(*
Signals are sent only once.
In order to resend the same signal, a global or a local reset is necessary.
*)
FUNCTION_BLOCK SignalHandling EXTENDS ExceptionHandling IMPLEMENTS I_SignalHandling 
VAR_OUTPUT
END_VAR

VAR_STAT
	bResetSignals : BOOL;
	aSignals : ARRAY[1..cMaxNumSignals] OF ST_Signal;
	uiSignalCounter : UINT := 0;
END_VAR

VAR CONSTANT
	cMaxNumSignals : UINT := 200;
	aEmptySignals : ARRAY[1..cMaxNumSignals] OF ST_Signal;
END_VAR

SUPER^();

METHOD BuildSignal : ST_Signal
VAR_INPUT
	eSignal	: E_Signal;
END_VAR
BuildSignal.eSignal := eSignal;
BuildSignal.eSignalOrigin := getSignalOrigin;
BuildSignal.sTimestamp := SYSTEMTIME_TO_STRING(fbTime.systemTime);
END_METHOD

METHOD GenericReceive : BOOL
VAR_INPUT
	eSignal : E_Signal;
END_VAR
VAR
	i : UINT;
END_VAR
FOR i := 1 TO uiSignalCounter
DO

	IF aSignals[i].eSignal = eSignal
	THEN
		//Reset the signal now
		GenericReceive := TRUE;
		RETURN;
	END_IF
		
END_FOR
END_METHOD

{warning 'Eigenschaftenimplementierung hinzufügen'}
PROPERTY getSignal : ST_Signal
GET
VAR CONSTANT
	stEmptySignal : ST_Signal;
END_VAR
IF SignalAvailable()
THEN
	getSignal := aSignals[uiSignalCounter];
	aSignals[uiSignalCounter] := stEmptySignal;
	uiSignalCounter := uiSignalCounter - 1;
END_IF
END_GET
END_PROPERTY

PROPERTY getSignalOrigin : E_Origin
GET
getSignalOrigin := eOrigin;
END_GET
END_PROPERTY

METHOD GlobalReset 
VAR
	stEmptySignal : ST_Signal;
	i : UINT;
END_VAR
aSignals := aEmptySignals;
uiSignalCounter := 0;
END_METHOD

METHOD Receive : BOOL
VAR_INPUT
	eSignal : E_Signal;
	eSignalOrigin : E_Origin;
END_VAR
VAR
	i : UINT;
END_VAR
FOR i := 1 TO uiSignalCounter
DO

	IF aSignals[i].eSignal = eSignal
	AND_THEN aSignals[i].eSignalOrigin = eSignalOrigin
	THEN
		//Reset the signal now
		Receive := TRUE;
		RETURN;
	END_IF
		
END_FOR
END_METHOD

METHOD ResetSignal : BOOL
VAR_INPUT
	eSignal : E_Signal;
	eSignalOrigin : E_Origin;
END_VAR
VAR
	i , k: UINT;
	stEmptySignal : ST_Signal;
END_VAR
IF SignalAvailable()
THEN
	
	FOR i:= 1 TO uiSignalCounter 
	DO
		//Search for exception
		IF aSignals[i].eSignal = eSignal 
		AND_THEN aSignals[i].eSignalOrigin = eSignalOrigin
		THEN
			//If found delete it from the array and adjust it
			ResetSignal := TRUE;
			FOR k:= i TO uiSignalCounter-1
			DO
				aSignals[k] := aSignals[k+1];
			END_FOR
			aSignals[k+1] := stEmptySignal;
			uiSignalCounter := uiSignalCounter - 1;
		END_IF  
	END_FOR

END_IF
END_METHOD

METHOD Signal : BOOL
VAR_INPUT
	stSignal	: ST_Signal;
END_VAR
VAR
	i : UINT;
END_VAR
IF uiSignalCounter <= cMaxNumSignals
THEN
	//Check if signal has been already sent
	FOR i := 1 TO uiSignalCounter
	DO
	
		IF aSignals[i].eSignal = stSignal.eSignal
		AND_THEN aSignals[i].eSignalOrigin = stSignal.eSignalOrigin
		THEN
			RETURN;
		END_IF
			
	END_FOR
	
	uiSignalCounter := uiSignalCounter + 1;
	aSignals[uiSignalCounter] := stSignal;
	Signal := TRUE;
	
ELSE

	Signal := FALSE;
	
END_IF
END_METHOD

METHOD SignalAvailable : BOOL
SignalAvailable := uiSignalCounter > 0;
END_METHOD

END_FUNCTION_BLOCK

(* stored: Version 1.1.0.1, ProductVersion 3.1.4024.0
   POU SignalHandling: Id {2ab09956-4cc3-4975-9dc3-0010378d9e03}, SpecialFunc None
   Method BuildSignal: Id {996c1d09-304f-429e-9c0a-344ab9aac518}
   Method GenericReceive: Id {cd45dc76-7fdf-4b42-ae86-f98cde4d6aee}
   Property getSignal: Id {645eaa58-74c1-4972-8cc3-7d57aeead74c}
   Get Get: Id {f990f5e6-985b-433a-8c56-c1dbdd717da5}
   Property getSignalOrigin: Id {2b76968e-adac-4046-8344-c15ca7f5eee9}
   Get Get: Id {539bb983-ad21-4398-8d00-b693f24fbb3e}
   Method GlobalReset: Id {24c0c733-846f-4865-94aa-11be04cabf5c}
   Method Receive: Id {beb99fe9-0fbb-4492-93b6-031e70c74753}
   Method ResetSignal: Id {14b95dca-d717-48d8-b998-d6f2c04e85fa}
   Method Signal: Id {1c8c2b8a-bf66-4183-925b-41180ac1de40}
   Method SignalAvailable: Id {518ea478-6e53-4f65-83ff-d325740067c3} *)
